Yaskawa INFORM job: R1_W63-A1(120,-90)KM-OK.JBI

/JOB
//NAME R1_W63-A1(120,-90)KM-OK
///FOLDERNAME KRIS-SCIANA
//POS
///NPOS 40,40,0,3,0,0
///TOOL 0
///POSTYPE PULSE
///PULSE
C00000=-21526,-164536,-89902,40074,64113,11441
C00001=-50807,-128086,-85912,36897,58218,89099
C00002=-109362,-74488,-62418,35906,91039,75494
C00003=-124724,-68487,-44042,35497,94233,70111
C00004=-123415,-69746,-42444,35648,92356,70038
C00005=-123251,-70839,-42731,35659,91973,69981
C00006=-123049,-74392,-31190,35688,84559,67669
C00007=-123049,-73512,-29667,35709,84161,67540
C00008=-123049,-73665,-29932,35705,84231,67562
C00009=-123181,-77945,-31666,35727,83357,67227
C00010=-123070,-74426,-30247,35707,84080,67506
C00011=-140110,-60526,-9750,48006,94045,60221
C00012=-137188,-61195,-10057,49085,92521,60774
C00013=-140350,-60464,-9723,47916,94170,60176
C00014=-120458,-68554,-40195,36121,90502,70642
C00015=-122490,-66733,-42633,35881,93336,70738
C00016=-120040,-68208,-52251,16848,99464,64704
C00017=-144710,-62118,-50826,-4733,101007,56514
C00018=-146144,-66915,-50905,-4953,98514,56114
C00019=-149481,-73487,-42698,-5469,89905,55339
C00020=-149481,-72872,-41457,-5469,89459,55358
C00021=-149481,-72153,-40021,-5469,88944,55384
C00022=-149481,-72250,-40217,-5469,89014,55380
C00023=-150502,-75356,-41590,-5649,88197,55077
C00024=-149720,-73470,-41485,-5512,89150,55294
C00025=-116046,-72347,-53392,-19558,100119,51510
C00026=-118570,-49017,-38824,-5964,114139,-21461
C00027=-120548,-59882,-50784,6437,105886,-80369
C00028=-95436,-82209,-48769,-2805,87673,-72259
C00029=-129111,-76469,-36414,20235,88686,-88163
C00030=-120580,-30937,-14274,5047,117192,-79737
C00031=-120572,-31635,-15793,5081,117765,-79708
C00032=-70896,-53168,-21216,-15225,103778,-64060
C00033=-84821,-64144,-27154,-20268,98953,-68239
C00034=-108509,-72952,-31286,-27494,90551,-74942
C00035=-139858,-71580,-30716,-34071,79863,-83742
C00036=-152133,-67005,-28672,-35427,75986,-87374
C00037=-104672,-73696,-58323,-15927,99894,-75667
C00038=-70152,-150754,-121601,-8267,55280,-63973
C00039=-70212,-174956,-136944,-8243,-11274,-63993
BC00000=121998,847,1075175
BC00001=55535,15,1075175
BC00002=92341,15,1075175
BC00003=126711,15,1075175
BC00004=126711,15,1075175
BC00005=126711,15,1075175
BC00006=126711,15,1075175
BC00007=126711,15,1075175
BC00008=126711,15,1075175
BC00009=126711,15,1075175
BC00010=126711,15,1075175
BC00011=126711,15,1075175
BC00012=126711,15,1075175
BC00013=126711,15,1075175
BC00014=126711,15,1075175
BC00015=126711,15,1075175
BC00016=120613,15,1075175
BC00017=120613,15,1075175
BC00018=120613,15,1075175
BC00019=120613,15,1075175
BC00020=120613,15,1075175
BC00021=120613,15,1075175
BC00022=120613,15,1075175
BC00023=120613,15,1075175
BC00024=120613,15,1075175
BC00025=109196,15,1075175
BC00026=132857,15,1075175
BC00027=151811,15,1075175
BC00028=161090,15,1075175
BC00029=161090,15,1075175
BC00030=152736,15,1075175
BC00031=152736,15,1075175
BC00032=161090,15,1075175
BC00033=161090,15,1075175
BC00034=161003,15,1075175
BC00035=161003,15,1075175
BC00036=161003,15,1075175
BC00037=93957,15,1075175
BC00038=93957,15,1075175
BC00039=93957,15,1075173
///POSTYPE BASE
///RECTAN
///RCONF 0,0,0,0,1,0,0,0,0,0,0,0,0,0,0,0,0,0,0,0,0,0,0,0
P00006=2.006,1.622,-0.565,0.0000,0.0000,0.0000
P00021=0.073,2.058,-0.109,0.0000,0.0000,0.0000
P00022=2.006,1.622,-0.565,0.0000,0.0000,0.0000
//INST
///DATE 2025/06/06 08:58
///ATTR SC,RW
///GROUP1 RB1,BS1
NOP
'r1_W63-A1(120,-90)
'Path S1498
SFTOF
MOVJ C00000 BC00000 VJ=20.00
MOVJ C00001 BC00001 VJ=20.00
MOVJ C00002 BC00002 VJ=20.00
MOVJ C00003 BC00003 VJ=20.00
MOVJ C00004 BC00004 VJ=20.00
MOVL C00005 BC00005 V=333.3
MOVL C00006 BC00006 V=60.0
REFP 3 C00007 BC00007
CALL JOB:SEARCH-R1
SET P021 P006
SFTON P021
MOVL C00008 BC00008 V=60.0
REFP 3 C00009 BC00009
CALL JOB:SEARCH-R1
SET P021 P006
SFTON P021
MOVL C00010 BC00010 V=60.0
MOVL C00011 BC00011 V=60.0
REFP 3 C00012 BC00012
CALL JOB:SEARCH-R1
SET P021 P006
SFTON P021
MOVL C00013 BC00013 V=60.0
MOVL C00014 BC00014 V=100.0
MOVL C00015 BC00015 V=166.7
'Path S1499
SFTOF
MOVJ C00016 BC00016 VJ=20.00
MOVJ C00017 BC00017 VJ=20.00
MOVJ C00018 BC00018 VJ=20.00
MOVL C00019 BC00019 V=333.3
MOVL C00020 BC00020 V=60.0
REFP 3 C00021 BC00021
CALL JOB:SEARCH-R1
SET P022 P006
SFTON P022
MOVL C00022 BC00022 V=60.0
REFP 3 C00023 BC00023
CALL JOB:SEARCH-R1
SET P022 P006
SFTON P022
MOVL C00024 BC00024 V=60.0
MOVL C00025 BC00025 V=166.7
'Path W1500
SFTOF
SFTON P022
MOVJ C00026 BC00026 VJ=20.00
MOVJ C00027 BC00027 VJ=20.00
SFTON P021
CALL JOB:COFNIJ_DRUT
MOVL C00028 BC00028 V=333.3
'SPRAWDZIC
MOVL C00029 BC00029 V=100.0 PL=0
REFP 1 C00030 BC00030
REFP 2 C00031 BC00031
MACRO1 MJ#(0) ARGF7
ARCON
MOVL C00032 BC00032 V=11.7
MOVL C00033 BC00033 V=11.7
SFTON P022
MOVL C00034 BC00034 V=11.7
MOVL C00035 BC00035 V=11.7
MOVL C00036 BC00036 V=11.7
ARCOF
SFTOF
MOVL C00037 BC00037 V=100.0
MOVL C00038 BC00038 V=166.7
MOVJ C00039 BC00039 VJ=20.00
SFTOF
END
